(*********************************** G.D S.p.A. - Technical Department ***********************************
============= PROGRAM INFO ============
FOLDER:             TBD
MACHINES INVOLVED:  TBD 

============= DESCRIPTION =============
csp machine declaration

============= REVISIONS ===============
Date		Version	 	Author      	Description             
----------	-------		------------  	--------------------------------------------
2020/07/20 	0000.00	 	M.Peppo			Virtual Master axis that allows the Transport Depth,
										Shuttle Depth, and Discharge Depth AccUchange axes to stay in sync
										as each gears to the master.
										
**********************************************************************************************************)
(*$R process_ref := prc; $*)
PROGRAM csp_case_transport_accU_virtualMaster
VAR
	
	prc:											process;
	prc_path:										STRING;
	
	axis:											axis;

	not_in_position:								message;
	geared_group_dif_exceeded:						message;
	dif_transport_and_shuttle:						LREAL := 982.8;
	dif_transport_and_discharge:					LREAL := 805.6;
	
	master_redefined:								BOOL;

	disable_req:									BOOL:=FALSE;
	position_req_mm:								LREAL:=0.0;(*$P unit:= mm; $*)
	move_velocity_req_mms:							LREAL:=10.0;(*$P unit:= mm; $*)
	position_req_tolerance_mm:						LREAL:=0.2;	(*$P $*)
	
	axis_status:									axis_status_enum := AXIS_STATUS_PARAMETERS_START;(*$M $*)
	in_position:									BOOL:=FALSE;(*$M $*)	
	actual_position_mm:								LREAL:=0.0; (*$M unit:= mm; $*)
	axis_move_condition:							BOOL:=FALSE;
	
	fsm_status:										csp_case_transport_accU_virtualMaster_enum;(*$M $*)
	fsm_next_status:								csp_case_transport_accU_virtualMaster_enum;
	fsm_enable_condition:							BOOL:=FALSE;
	debug_state_machine:							BOOL:=FALSE;
	debug_state_machine_one_step:					BOOL:=FALSE;
	slave_follow_limit:								LREAL := 0.05;
	First_scan:										BOOL := TRUE;
	JogEnableRTRIG:									R_Trig;
	JogActive:										BOOL;
	
	debug1: DINT;
END_VAR

_read_var_input();

_object_manager();

IF NOT objects_running()
THEN
	RETURN;	
END_IF

_read_process_image();

_mode_manager();

CASE process_get_mode(prc) OF
	MODE_ABSENT,
	MODE_INACTIVE:
		RETURN;
	MODE_TEST:
		_handle_process_test();
END_CASE

_set_runtime_properties();

(********************************* BODY *********************************)

//Axis move condition
IF 	csp_main_accuChange.case_transport_accU_depth_move_req
	OR jog_manager_is_jog_axis_active(SMTR61210_SMTR61200_SMTR61420_CASE_FEED_SHUTTLE_TRANSPORT_AND_DISCHARGE_DEPTH, csp_main_jogManager.jog_manager_accuchange)
THEN
	axis_move_condition := TRUE;
ELSE
	axis_move_condition := FALSE;
END_IF

JogActive := jog_manager_is_jog_axis_active(SMTR61210_SMTR61200_SMTR61420_CASE_FEED_SHUTTLE_TRANSPORT_AND_DISCHARGE_DEPTH, csp_main_jogManager.jog_manager_accuchange);

JogEnableRTRIG(CLK := JogActive);

(*Jog Mode - Redefine Position*)
IF JogEnableRTRIG.Q
	//AND (axis_is_standstill(axis) or axis_is_position_redefined(axis))
	//AND ABS(actual_position_mm - csp_case_transport_accU_depth.actual_position_mm) > 0.5
	OR First_scan
THEN
	axis_redefine_position (
		position    :=  csp_case_transport_accU_depth.actual_position_mm,
		mode        :=  AXIS_REDEFINE_POSITION_MODE_ABSOLUTE,
		CONVERSION_this        :=  AXIS);	
END_IF

IF jog_manager_is_jog_axis_active(SMTR61210_SMTR61200_SMTR61420_CASE_FEED_SHUTTLE_TRANSPORT_AND_DISCHARGE_DEPTH, csp_main_jogManager.jog_manager_accuchange)
	AND NOT axis_is_standstill(axis)
	AND 
	(
	(ABS(axis_get_following_error(csp_case_feed_shuttle_accu_Depth.axis)) > slave_follow_limit)
	OR
	(ABS(axis_get_following_error(csp_case_feed_reject_accU_depth.axis)) > slave_follow_limit)
	OR
	(ABS(axis_get_following_error(csp_case_transport_accu_depth.axis)) > slave_follow_limit)
	OR
		(
			(
			NOT axis_is_gear_engaged(csp_case_feed_shuttle_accu_Depth.axis)
			OR 
			NOT axis_is_gear_engaged(csp_case_feed_reject_accU_depth.axis)	
			OR 
			NOT axis_is_gear_engaged(csp_case_transport_accu_depth.axis)
			)
		AND debug1.1
		)	
	)
THEN
	axis_stop(
		deceleration 	:= csp_main_accuChange.CONSTANTS.MAX_DECELERATION_MMpSEC2 * 0.5,
		jerk 			:= csp_main_accuChange.CONSTANTS.MAX_JERK_MMpSEC3,
		CONVERSION_this 			:= axis);
	debug1.2 := TRUE;
END_IF

(*FSM Control*)
fsm_enable_condition := axis_is_ok(FALSE, axis)
						(*AND
						process_is_ready(prc) *)
						AND
						process_subtree_is_ready(prc)
						AND
						process_get_mode(csp_main_accuChange.prc) = MODE_OPERATIONAL
						AND
						axis_move_condition
						AND
						NOT jog_manager_is_jog_axis_active(SMTR61210_SMTR61200_SMTR61420_CASE_FEED_SHUTTLE_TRANSPORT_AND_DISCHARGE_DEPTH, csp_main_jogManager.jog_manager_accuchange)
						AND
						NOT disable_req;	
					
IF	(NOT fsm_enable_condition
	OR
	disable_req)
	AND
	fsm_status <> CSP_CASE_TRANSPORT_ACCU_VIRTUAL_MASTER_STATUS_DISABLED
	AND
	fsm_status < CSP_CASE_TRANSPORT_ACCU_VIRTUAL_MASTER_STATUS_STOP_REQUEST
THEN
	fsm_status	:=	CSP_CASE_TRANSPORT_ACCU_VIRTUAL_MASTER_STATUS_STOP_REQUEST;
END_IF


CASE fsm_status OF
	
	CSP_CASE_TRANSPORT_ACCU_VIRTUAL_MASTER_STATUS_NOT_INITIALIZED:
	
        IF	axis_is_ok(return_when_absent := TRUE, CONVERSION_this := axis)
        THEN
            fsm_next_status := CSP_CASE_TRANSPORT_ACCU_VIRTUAL_MASTER_STATUS_DISABLED;
        END_IF

		
	CSP_CASE_TRANSPORT_ACCU_VIRTUAL_MASTER_STATUS_DISABLED:
	
		master_redefined := FALSE;
	
		IF	fsm_enable_condition
		THEN
			(* Axis with absolute encoder, no home procedure request *)
			fsm_next_status := CSP_CASE_TRANSPORT_ACCU_VIRTUAL_MASTER_STATUS_POSITION_CHECK;
		END_IF;
	
		
	CSP_CASE_TRANSPORT_ACCU_VIRTUAL_MASTER_STATUS_POSITION_CHECK:

		(* CHECKS IF AXIS IS IN TOLERANCE *)
		IF 	NOT csp_case_transport_accu_depth.in_position
			AND machine_is_ready(csp.mch)  
		THEN
			(* NOT IN TOLERANCE - NEED TO GEAR AND MOVE *)
			fsm_next_status := CSP_CASE_TRANSPORT_ACCU_VIRTUAL_MASTER_STATUS_ENABLE_REQUEST;
		END_IF		
		
		
	CSP_CASE_TRANSPORT_ACCU_VIRTUAL_MASTER_STATUS_ENABLE_REQUEST:
	
		axis_enable(axis);
		IF axis_is_standstill(axis)
		THEN
			IF axis_redefine_position (
				position    :=  csp_case_transport_accU_depth.actual_position_mm,
				mode        :=  AXIS_REDEFINE_POSITION_MODE_ABSOLUTE,
				CONVERSION_this        :=  AXIS)
			THEN
				master_redefined := TRUE;
				fsm_next_status	:=	CSP_CASE_TRANSPORT_ACCU_VIRTUAL_MASTER_STATUS_CHECK_SLAVE_GEAR;
			END_IF
		END_IF	
		
			
	CSP_CASE_TRANSPORT_ACCU_VIRTUAL_MASTER_STATUS_CHECK_SLAVE_GEAR:
	
		IF axis_is_gear_engaged(csp_case_feed_shuttle_accu_depth.axis)
			AND axis_is_gear_engaged(csp_case_transport_accu_depth.axis)
			AND axis_is_gear_engaged(csp_case_feed_reject_accU_depth.axis)
		THEN
			fsm_next_status := CSP_CASE_TRANSPORT_ACCU_VIRTUAL_MASTER_STATUS_ENABLED;
		END_IF
	
		
	CSP_CASE_TRANSPORT_ACCU_VIRTUAL_MASTER_STATUS_ENABLED:
	
		IF axis_move_condition 
		THEN
			fsm_next_status	:= CSP_CASE_TRANSPORT_ACCU_VIRTUAL_MASTER_STATUS_ABS_MOVE_REQUEST;	
		END_IF
		
		
	CSP_CASE_TRANSPORT_ACCU_VIRTUAL_MASTER_STATUS_ABS_MOVE_REQUEST:

		IF	axis_is_position_redefined(axis)
		THEN
			 axis_move_absolute(
				position 		:= csp_case_transport_accU_depth.position_req_mm,
				velocity 		:= csp_case_transport_accU_depth.move_velocity_req_mms,
				direction		:= AXIS_SHORTEST_WAY,
				acceleration 	:= csp_main_accuChange.CONSTANTS.MAX_ACCELERATION_MMpSEC2 * 0.1,
				deceleration 	:= csp_main_accuChange.CONSTANTS.MAX_DECELERATION_MMpSEC2 * 0.1,
				jerk 			:= csp_main_accuChange.CONSTANTS.MAX_JERK_MMpSEC3, 
				buffer_mode 	:= AXIS_BUFFER_MODE_BUFFERED,
				CONVERSION_this := axis
				); 
				
			fsm_next_status	:=	CSP_CASE_TRANSPORT_ACCU_VIRTUAL_MASTER_STATUS_ABS_MOVING;
		END_IF

		
	CSP_CASE_TRANSPORT_ACCU_VIRTUAL_MASTER_STATUS_ABS_MOVING:

		IF axis_is_standstill(axis)
			OR (ABS(axis_get_following_error(csp_case_feed_shuttle_accu_Depth.axis)) > slave_follow_limit)
			OR (ABS(axis_get_following_error(csp_case_feed_reject_accU_depth.axis)) > slave_follow_limit)
			OR (ABS(axis_get_following_error(csp_case_transport_accu_depth.axis)) > slave_follow_limit)
			OR
			(
				axis_is_moving(axis)
			AND 
				(
				NOT axis_is_moving(csp_case_feed_shuttle_accu_Depth.axis)
				OR NOT axis_is_moving(csp_case_feed_reject_accU_depth.axis)
				OR NOT axis_is_moving(csp_case_transport_accu_depth.axis)
				)
			)
		THEN
			fsm_next_status := CSP_CASE_TRANSPORT_ACCU_VIRTUAL_MASTER_STATUS_STOP_REQUEST;//CSP_CASE_TRANSPORT_ACCU_VIRTUAL_MASTER_STATUS_DISABLE_REQUEST;
		END_IF
		
		
	CSP_CASE_TRANSPORT_ACCU_VIRTUAL_MASTER_STATUS_STOP_REQUEST:

		axis_stop(
		    deceleration 	:= csp_main_accuChange.CONSTANTS.MAX_DECELERATION_MMpSEC2 * 0.5,
		    jerk 			:= csp_main_accuChange.CONSTANTS.MAX_JERK_MMpSEC3,
		    CONVERSION_this 			:= axis);

		IF 	axis_is_standstill(axis)
			OR
			NOT axis_is_ok(FALSE, axis)
			OR
			axis_is_disabled(axis)
		THEN
			fsm_next_status := CSP_CASE_TRANSPORT_ACCU_VIRTUAL_MASTER_STATUS_DISABLE_REQUEST;
		END_IF

		
	CSP_CASE_TRANSPORT_ACCU_VIRTUAL_MASTER_STATUS_DISABLE_REQUEST:
   		axis_disable(axis);
        IF	axis_is_disabled(axis)
        THEN
            fsm_next_status := CSP_CASE_TRANSPORT_ACCU_VIRTUAL_MASTER_STATUS_DISABLED;
        END_IF;

END_CASE;

IF NOT debug_state_machine
	OR
	debug_state_machine_one_step
THEN
	fsm_status := fsm_next_status;
	debug_state_machine_one_step := FALSE;
END_IF

(* Axes engaged for jog management *)
jog_manager_set_all_slave_axis_engaged(
	index					:= SMTR61210_SMTR61200_SMTR61420_CASE_FEED_SHUTTLE_TRANSPORT_AND_DISCHARGE_DEPTH, 
	all_slave_axis_engaged	:= axis_is_gear_engaged(csp_case_feed_shuttle_accU_depth.axis) AND axis_is_gear_engaged(csp_case_transport_accU_depth.axis) AND axis_is_gear_engaged(csp_case_feed_reject_accU_depth.axis),							   								 	
	CONVERSION_this			:= csp_main_jogManager.jog_manager_accuchange);
	
	
First_scan := FALSE;
(************************************************************************)

_handle_messages();

_write_output();

ACTION _handle_messages:
IF (ABS(csp_case_transport_accU_depth.actual_position_mm - csp_case_feed_shuttle_accU_depth.actual_position_mm) - dif_transport_and_shuttle) < 0.5
	AND (ABS(csp_case_transport_accU_depth.actual_position_mm - csp_case_feed_reject_accU_depth.actual_position_mm) - dif_transport_and_discharge) < 0.5
THEN
	process_message_reset(geared_group_dif_exceeded);
END_IF
END_ACTION

ACTION _handle_process_test:
;
END_ACTION

ACTION _mode_manager:
IF process_mode_req_is_pending(prc)
THEN
    process_apply_mode_req_first_step(prc);
    CASE process_get_mode(prc) OF
        MODE_TO_ABSENT:
			;
        MODE_TO_INACTIVE:
			;
        MODE_TO_TEST:
			;
        MODE_TO_OPERATIONAL:
			;
    END_CASE
    process_apply_mode_req_second_step(prc);
END_IF
END_ACTION

ACTION _object_manager:
IF objects_initialization()
THEN
	sub_process_init(
		object_name								:= 'csp_case_transport_accU_virtualMaster.prc', 
		process									:= csp_case_transport_accU.prc, 
		CONVERSION_this							:= prc);
		
	prc_path 									:= process_get_path(prc);
	
	axis_init(
		object_name 							:= CONCAT(prc_path, '_axis'),
		axis_type 								:= AXIS_TYPE_VIRTUAL,
		encoder_scaling_factor 					:= G_VIRTUAL_ENCODER_SCALING_FACTOR_DEGPINC,
		modulo 									:= 1024,
		process 								:= prc,
		CONVERSION_this 						:= axis);
		
	axis_set_rotation_direction(
		invert_encoder_counting					:= FALSE,
		invert_motor_polarity					:= FALSE,
		CONVERSION_this							:= axis);
	
	axis_set_max_dynamic(
		reference_velocity						:=	csp_main_accuChange.CONSTANTS.MAX_VELOCITY_MMpSEC,
		velocity								:=	csp_main_accuChange.CONSTANTS.MAX_VELOCITY_MMpSEC,
		acceleration							:=	csp_main_accuChange.CONSTANTS.MAX_ACCELERATION_MMpSEC2,
		deceleration							:=	csp_main_accuChange.CONSTANTS.MAX_DECELERATION_MMpSEC2,
		jerk									:=	csp_main_accuChange.CONSTANTS.MAX_JERK_MMpSEC3,
		following_error							:=	csp_main_accuChange.CONSTANTS.MAX_FOLLOWING_ERROR_MM,
		CONVERSION_this							:=	axis);
	
	jog_manager_add_axis(
		list_index								:= SMTR61210_SMTR61200_SMTR61420_CASE_FEED_SHUTTLE_TRANSPORT_AND_DISCHARGE_DEPTH,
		axis									:= axis,
		master_axis								:= TRUE,
		jog_type								:= JOG_TYPE_LINEAR,
		sw_limit_positive						:= 30,
		sw_limit_negative						:= 0,
		CONVERSION_this							:= csp_main_jogManager.jog_manager_accuchange);
		
	process_message_init(
		object_name:= CONCAT(prc_path, '_geared_group_dif_exceeded'), 
		behaviour:= MESSAGE_BEHAVIOUR_STATE, 
		reset_timeout:= 0, 
		disableable:= TRUE, 
		individual_reset:= FALSE, 
		machine_reaction:= MACHINE_REACTION_NO_STOP,
		typology:=  MESSAGE_TYPOLOGY_NOT_VISIBLE,
		process:= prc, 
		CONVERSION_this:= geared_group_dif_exceeded);
	
END_IF

IF objects_running()
THEN
	process_cycle(prc);
	axis_cycle(axis);
END_IF
END_ACTION

ACTION _read_process_image:
;
END_ACTION

ACTION _read_var_input:
disable_req := csp_case.disable_req;
END_ACTION

ACTION _set_runtime_properties:
axis_status := axis_get_status(axis);
actual_position_mm :=axis_get_actual_incremental_position(axis); (* axis_get_actual_modulo_position(axis); only with modulo*)

IF ABS(position_req_mm - actual_position_mm)< position_req_tolerance_mm
	OR
	process_get_mode(prc)= MODE_ABSENT
	OR
	process_get_mode(csp_main_accuChange.prc) = MODE_ABSENT
THEN
	in_position := TRUE;
ELSE
	in_position := TRUE; //AMR //set to false when ready	
END_IF
END_ACTION

ACTION _write_output:
;
END_ACTION

END_PROGRAM

(* stored: Version 1.1.0.1, ProductVersion 3.1.4024.3
   POU csp_case_transport_accU_virtualMaster: Id {c8ad2737-0e7c-4bc3-92d9-4cff5e72ba7d}, SpecialFunc None
   Action _handle_messages: Id {8e28a825-4819-40b2-896f-43a88560a12e}
   Action _handle_process_test: Id {fc493a26-b0c2-4037-b211-f4c992275ebf}
   Action _mode_manager: Id {8f14e057-9a79-44ff-a729-4160aa47fc19}
   Action _object_manager: Id {1ddfd718-8124-4598-9369-f64e8f4581aa}
   Action _read_process_image: Id {49149458-15fc-4e54-81a1-2a5252902412}
   Action _read_var_input: Id {e9759bbe-8a83-4248-94a5-5c2aa5d0d288}
   Action _set_runtime_properties: Id {e5355189-b1ee-420c-aa48-0fa8fd029acf}
   Action _write_output: Id {26918356-7be3-451c-83f0-8b0b23a135f7} *)
